// TIA Portal V19 export
TYPE "lexchangetray_typeplasticWorkStation_signalTM_Simulation"
// Type: Bool
// stored: Access Published
   STRUCT
      inspectionAfterPlasticTrayJacking : Bool;   // Manual mode parameters for axis control interface
      inspectionBeforePlasticTrayJacking : Bool;   // Manual mode parameters for axis control interface
      plasticTrayFeedingDetection : Bool;   // Manual mode parameters for axis control interface
      plasticTrayLiftingCylinderHomePositionDetection1 : Bool;   // Manual mode parameters for axis control interface
      plasticTrayTrayInplaceDetection : Bool;   // Manual mode parameters for axis control interface
      plasticTrayLiftingCylinderWorkingPositionDetection1 : Bool;   // Manual mode parameters for axis control interface
      scapegoatSignal1 : Bool;   // Manual mode parameters for axis control interface
      scapegoatSignal2 : Bool;   // Manual mode parameters for axis control interface
   END_STRUCT;
END_TYPE
